FUNCTION_BLOCK FB_Axis EXTENDS FB_Base IMPLEMENTS ITF_0_BaseComponent
VAR_INPUT
END_VAR
VAR_OUTPUT
END_VAR
VAR
END_VAR

METHOD M_activate : BOOL
VAR_INPUT
END_VAR
END_METHOD

METHOD M_cleanup : BOOL
VAR_INPUT
END_VAR
END_METHOD

METHOD M_configure : BOOL
VAR_INPUT
END_VAR
END_METHOD

METHOD M_deactivate : BOOL
VAR_INPUT
END_VAR
END_METHOD

METHOD M_destroy : BOOL
VAR_INPUT
END_VAR
END_METHOD

METHOD M_shutdown : BOOL
VAR_INPUT
END_VAR
END_METHOD

METHOD onActivate : BOOL
VAR_INPUT
END_VAR
END_METHOD

METHOD onCleanup : BOOL
VAR_INPUT
END_VAR
END_METHOD

METHOD onConfigure : BOOL
VAR_INPUT
END_VAR
END_METHOD

METHOD onDeactivate : BOOL
VAR_INPUT
END_VAR
END_METHOD

METHOD onError : BOOL
VAR_INPUT
END_VAR
END_METHOD

METHOD onShutdown : BOOL
VAR_INPUT
END_VAR
END_METHOD

PROPERTY P_ID : UINT
GET
END_GET
SET
END_SET
END_PROPERTY

PROPERTY P_Name : String
GET
END_GET
END_PROPERTY

PROPERTY P_Path : String
GET
END_GET
END_PROPERTY

PROPERTY P_State : eState
GET
END_GET
SET
END_SET
END_PROPERTY

END_FUNCTION_BLOCK

(* stored: Version 1.1.0.1, ProductVersion 3.1.4026.18
   POU FB_Axis: Id {9e4ffeba-a891-443c-b3e5-b3f139fd35fe}, SpecialFunc None
   Folder Activities: Id {06120b37-9249-40c4-9170-129c2634ed82}
   Folder Transitions: Id {017e141b-1342-4c67-8ad7-1808f1bdbc4f}
   Method M_activate: Id {54e6b466-4a12-4074-b465-d0b8e8c3558c}
   Method M_cleanup: Id {e91931c4-06bd-469c-a7d8-79ded78b6d98}
   Method M_configure: Id {d9630fbb-4cd2-47d1-8fc5-a5a6051e6304}
   Method M_deactivate: Id {699be2d0-36cb-4504-ae20-389e3df7cff6}
   Method M_destroy: Id {cc3501d8-1c5a-47c1-b5f3-768d8d9ccf3f}
   Method M_shutdown: Id {da7031a9-84a2-438c-b578-d0c80904a5d5}
   Method onActivate: Id {dff9d669-6f40-4f00-90d9-3787e79ba4a4}
   Method onCleanup: Id {80fa50ea-abbc-41d9-a37b-59c86da9d595}
   Method onConfigure: Id {9c8ee034-539b-4679-a220-e9e172d34c39}
   Method onDeactivate: Id {7b5bbaf4-d2cc-4310-8122-de7176198651}
   Method onError: Id {9a005bfb-be70-4cfa-9cc0-3bf4840f8b47}
   Method onShutdown: Id {a3cf4dc0-c49b-489c-8e1e-811c54f2901e}
   Property P_ID: Id {64850be6-4d1e-47ed-bf29-aaed00838e9f}
   Get Get: Id {01aa5cf0-2fe2-448d-a4b0-3fd79cc979f8}
   Set Set: Id {af160821-6079-4445-9de3-8861626924b5}
   Property P_Name: Id {93487327-35e4-4087-bb5d-98718c2d7005}
   Get Get: Id {a9078179-15d7-4493-94d2-86a0cd11f892}
   Property P_Path: Id {e999ff4c-5501-4405-953a-f17558d3540c}
   Get Get: Id {6f2ac6a8-bc2f-4f24-b31e-d4e086fc26f3}
   Property P_State: Id {ccc67b2c-b422-47eb-90b2-34d846e9d8c2}
   Get Get: Id {fa198063-5954-4506-853c-5eeee5c0e776}
   Set Set: Id {92804267-2cf0-40f8-8756-0848ad65104a} *)
